// TIA Portal V17 export
// export: Created 2026-04-13T11:12:42.0535092Z, ExportSetting WithDefaults, DisplayName Totally Integrated Automation Portal, DisplayVersion V17 Update 4, DisplayName TIA Portal Openness, DisplayVersion V17 Update 4, DisplayName TIA Portal Version Control Interface, DisplayVersion V17, DisplayName SINAMICS Startdrive Advanced, DisplayVersion V17, DisplayName SINAMICS Startdrive G130, G150, S120, S150, SINAMICS MV, S210, DisplayVersion V17, DisplayName SINAMICS Startdrive G110M, G120, G120C, G120D, G120P, G115D, DisplayVersion V17, DisplayName STEP 7 Professional, DisplayVersion V17 Update 4, DisplayName STEP 7 Safety, DisplayVersion V17, DisplayName WinCC Professional, DisplayVersion V17 Update 4
FUNCTION_BLOCK "斜坡函数发生器"   // FB85, SCL
{ S7_Optimized_Access := 'TRUE' }
VERSION : 0.1
// stored: AutoNumber true, IsIECCheckEnabled false, IsRetainMemResEnabled false, MemoryReserve 100, SetENOAutomatically false, UDAEnableTagReadback false
   VAR_INPUT
      输入 : Real;
      斜坡激活 : Bool;   // 0：直接输出 1：斜坡输出
      上升斜率 : Real := 1.0;   // 斜坡上升增量值 （单位值/秒）
      下降斜率 : Real := 1.0;   // 斜坡下降增量值 （ 单位值/秒）
      输出上限 : Real := 100.0;
      输出下限 : Real := 0.0;
   END_VAR
   VAR_OUTPUT
      输出 : Real;
   END_VAR
BEGIN

   //可用于电机的速度给定以实现平滑升/降速；重要的调节阀门设定，进行平滑过度，防止水锤及工艺扰动等现象
   //在循环中断OB30中调用该FB块，OB30循环时间设置为100ms。
   //如果上升斜率设置为1/s，输入则上升斜坡将持续10s（设定值从0增加至10）。
   //公式：Y=Y+A。

   IF NOT #斜坡激活 THEN
       //直接输出
       #输出 := #输入;
   ELSE
       //斜坡输出
       IF #输入 > #输出 THEN
           //斜坡上升
           #输出 := #输出 + #上升斜率 / 10.0;
       END_IF;
       IF #输入 < #输出 THEN
           //斜坡下降
           #输出 := #输出 - #下降斜率 / 10.0;
       END_IF;
   END_IF;


   //输出限幅
   IF #输出 > #输出上限 THEN
       #输出 := #输出上限;
   END_IF;
   IF #输出 < #输出下限 THEN
       #输出 := #输出下限;
   END_IF;
END_FUNCTION_BLOCK
